FUNCTION_BLOCK FB_OuterCapillaryTubeMats EXTENDS FB_SystemContinous
VAR_INPUT
	stAmbientState : ST_AmbientState;
END_VAR
VAR_OUTPUT
END_VAR
VAR
	//default parameters
	localDefaultParameters : ST_OuterCapillaryTubeMatsDefaultParameters;	
	
	//pumps
	stPU235DefaultParameters : ST_PumpGrundfosMagna3DefaultParameters;
	stPU600DefaultParameters : ST_PumpGrundfosMagna3DefaultParameters;
	
	PU235 : FB_PumpGrundfosMagna3 := (ST_DefaultParameters := stPU235DefaultParameters);
	PU600 : FB_PumpGrundfosMagna3 := (ST_DefaultParameters := stPU600DefaultParameters);	
	PU690 : FB_Pump2Point; //CM pump (storage side)
	
	//valves
	stSV235DefaultParameters : ST_DiscreteValveDefaultParameters := (nFeedback := 0);
	stSV605DefaultParameters : ST_DiscreteValveDefaultParameters := (nFeedback := 3);
	stRV600DefaultParameters : ST_MixingValveDefaultParameters := (bFeedbackSignal := FALSE, tTaskCycleTime := GlobalVariables.tCtrlCycleTime_MAIN, tCtrlCycleTime := GlobalVariables.tCtrlCycleTime_MAIN);	
	stRV640DefaultParameters : ST_MixingValveDefaultParameters := (bFeedbackSignal := FALSE, tTaskCycleTime := GlobalVariables.tCtrlCycleTime_MAIN, tCtrlCycleTime := GlobalVariables.tCtrlCycleTime_MAIN);
	stRV660DefaultParameters : ST_MixingValveDefaultParameters := (bFeedbackSignal := FALSE, tTaskCycleTime := GlobalVariables.tCtrlCycleTime_MAIN, tCtrlCycleTime := GlobalVariables.tCtrlCycleTime_MAIN);
	
	SV235 : FB_DiscreteValve := (ST_DefaultParameters := stSV235DefaultParameters);
	SV605 : FB_DiscreteValve := (ST_DefaultParameters := stSV605DefaultParameters);
	RV600 : FB_MixingValve := (ST_DefaultParameters := stRV600DefaultParameters);
	RV640 : FB_MixingValve := (ST_DefaultParameters := stRV640DefaultParameters); //east
	RV660 : FB_MixingValve := (ST_DefaultParameters := stRV660DefaultParameters); //west
	
	//sensors
	WMZ235 : FB_MollineC3HeatCounter;
	
	//internal variables
	bSetStatusOn_PU235 	: BOOL;
	bSetStatusOn_PU600 	: BOOL;
	bSetStatusOn_PU690 	: BOOL;
	bSetStatusOn_SV235 	: BOOL;	
	bSetStatusOn_RV600 	: BOOL;
	bSetStatusOn_RV640 	: BOOL;
	fSetPoint_RV640 	: REAL;
	bSetStatusOn_RV660 	: BOOL;
	fSetPoint_RV660 	: REAL;
	
	//clock and timer
	stDefaultParameters_Clock : ST_ClockDefaultParameters := (tTaskCycleTime := GlobalVariables.tCtrlCycleTime_MAIN, tCtrlCycleTime := T#1M);
	Clock : FB_Clock := (ST_DefaultParameters := stDefaultParameters_Clock);
	bStartTimer : BOOL;
	Timer : TON;
END_VAR

MAIN();
//use timer because valve has no feedback signal (75 sec)
Timer(IN := bStartTimer,
	PT := T#75S);
Clock();

//pumps
PU235.GetState_Profibus();
PU235(bSetStatusOnAutomatic := bSetStatusOn_PU235,
	fSetPointAutomatic := 70,
	bAlgorithmPermission := bAlgorithmPermission,
	nControlModeAutomatic := 0);
PU235.SetState_Profibus();

//use AUTO-Adapt control mode
PU600.GetState_Profibus();
PU600(bSetStatusOnAutomatic := bSetStatusOn_PU600,
	fSetPointAutomatic := 70,
	bAlgorithmPermission := bAlgorithmPermission,
	nControlModeAutomatic := 0);
PU600.SetState_Profibus();

PU690(bSetStatusOnAutomatic := bSetStatusOn_PU690,
	bAlgorithmPermission := bAlgorithmPermission);
PU690.SetState_BO();

//valves
SV235.GetState_BI();
SV235(bSetStatusOnAutomatic := bSetStatusOn_SV235,
	bAlgorithmPermission := bAlgorithmPermission);
SV235.SetState_BO();

SV605.GetState_BI();
SV605(bSetStatusOnAutomatic := TRUE,
	bAlgorithmPermission := bAlgorithmPermission);
SV605.SetState_BO();

//RV600 uses heating mode to control inlet temperature into PWT6 (with temperature difference of 7 K of primary and secondary side)
RV600.GetState_AI();
RV600(bSetStatusOnAutomatic := bSetStatusOn_RV600,
	fSetPointAutomatic := fSetPoint,
	bAlgorithmPermission := bAlgorithmPermission,
	fTemperatureExternal := PU235.fTemperatureExternal,
	nControlModeAutomatic := 2);
RV600.SetState_AO();

RV640.GetState_AI();
RV640(bSetStatusOnAutomatic := bSetStatusOn_RV640,
	fSetPointAutomatic := fSetPoint_RV640,
	bAlgorithmPermission := bAlgorithmPermission,
	nControlModeAutomatic := 0);
RV640.SetState_AO();

RV660.GetState_AI();
RV660(bSetStatusOnAutomatic := bSetStatusOn_RV660,
	fSetPointAutomatic := fSetPoint_RV660,
	bAlgorithmPermission := bAlgorithmPermission,
	nControlModeAutomatic := 0);
RV660.SetState_AO();

//insert heat counter telegramm from other task
WMZ235();

METHOD AmbientControl : BOOL
VAR_INPUT
END_VAR
//check for rain
IF NOT stAmbientState.bRain THEN
	bSetStatusOn_PU690 := TRUE;
ELSE
	bSetStatusOn_PU690 := FALSE;
END_IF

//check for time
IF Clock.stClockState.fHour < 12 THEN
	//use west facade	
	fSetPoint_RV640 := 100;
	fSetPoint_RV660 := 0;
ELSE
	//use east facade
	fSetPoint_RV640 := 0;
	fSetPoint_RV660 := 100;
END_IF
END_METHOD

METHOD PROTECTED  CheckError : BOOL
VAR_INPUT
END_VAR
VAR_OUTPUT
	bError : BOOL;
END_VAR
VAR
	bError_PU235 : BOOL;
	bError_PU600 : BOOL;
	bError_SV235 : BOOL;
END_VAR
//check pumps for errors
bError_PU235 := PU235.bError;
bError_PU600 := PU600.bError;

//check valve SV235 for an error
IF SV235.bStatusOn AND PU235.bStatusOn THEN
	bError_SV235 := TRUE;
END_IF

bError := bError_PU235 OR bError_PU600 OR bError_SV235;
END_METHOD

METHOD PROTECTED  Operational : BOOL
VAR_INPUT
END_VAR
VAR_OUTPUT
	bSwitchToWorking : BOOL := FALSE;
END_VAR
bSetStatusOn_PU235 := TRUE;
bSetStatusOn_PU600 := TRUE;
AmbientControl();

IF PU235.bStatusOn AND PU600.bStatusOn THEN
	bSwitchToWorking := TRUE;
END_IF;
END_METHOD

METHOD PROTECTED  RampDown : BOOL
VAR_INPUT
END_VAR
VAR_OUTPUT
	bRampDownFinished : BOOL := FALSE;
END_VAR
bSetStatusOn_PU600 := FALSE;
bSetStatusOn_PU235 := FALSE;
bSetStatusOn_PU690 := FALSE;
bSetStatusOn_SV235 := FALSE;
bSetStatusOn_RV600 := FALSE;
bSetStatusOn_RV640 := FALSE;
bSetStatusOn_RV660 := FALSE;
bStartTimer := TRUE;

IF Timer.Q THEN
	bRampDownFinished := TRUE;
	bStartTimer := FALSE;
END_IF
END_METHOD

METHOD PROTECTED  RampUp : BOOL
VAR_INPUT
END_VAR
VAR_OUTPUT
	bRampUpFinished : BOOL := FALSE;
END_VAR
bSetStatusOn_SV235 := TRUE;
bSetStatusOn_RV600 := TRUE;
bSetStatusOn_RV640 := TRUE;
bSetStatusOn_RV660 := TRUE;
bStartTimer := TRUE;

IF Timer.Q THEN
	bRampUpFinished := TRUE;
	bStartTimer := FALSE; //resets timer
END_IF

//check for rain
AmbientControl();
END_METHOD

METHOD PROTECTED   SetSetPointLimits : BOOL
VAR_INPUT
END_VAR
aSetPointLimits[1] := localDefaultParameters.aSetPointLimitsTemperature[1];
aSetPointLimits[2] := localDefaultParameters.aSetPointLimitsTemperature[2];
END_METHOD

METHOD PROTECTED  Working : BOOL
VAR_INPUT
END_VAR
VAR_OUTPUT
	bSwitchToOperational : BOOL := FALSE;
END_VAR
AmbientControl();
END_METHOD

END_FUNCTION_BLOCK

(* stored: Version 1.1.0.1, ProductVersion 3.1.4024.10
   POU FB_OuterCapillaryTubeMats: Id {f8d40369-147e-4cbe-aff1-5204bfee2138}, SpecialFunc None
   Method AmbientControl: Id {88a15c5a-66ea-4cac-bc26-6cc439e986de}
   Method CheckError: Id {b5c5e5e8-42f6-4651-a2ed-f1d07717775f}
   Method Operational: Id {c5d251a1-4b82-443d-8a1b-17b15e56f92c}
   Method RampDown: Id {a23ccce8-0424-4b4c-82c7-de0b91fea1cb}
   Method RampUp: Id {a529c9d9-81e0-4127-865c-b1ad3753334d}
   Method SetSetPointLimits: Id {7fcac2fe-640f-418c-9c40-05dd5101cb8c}
   Method Working: Id {38cc873a-2ab0-456c-a4f7-7981cf3fbe46} *)
